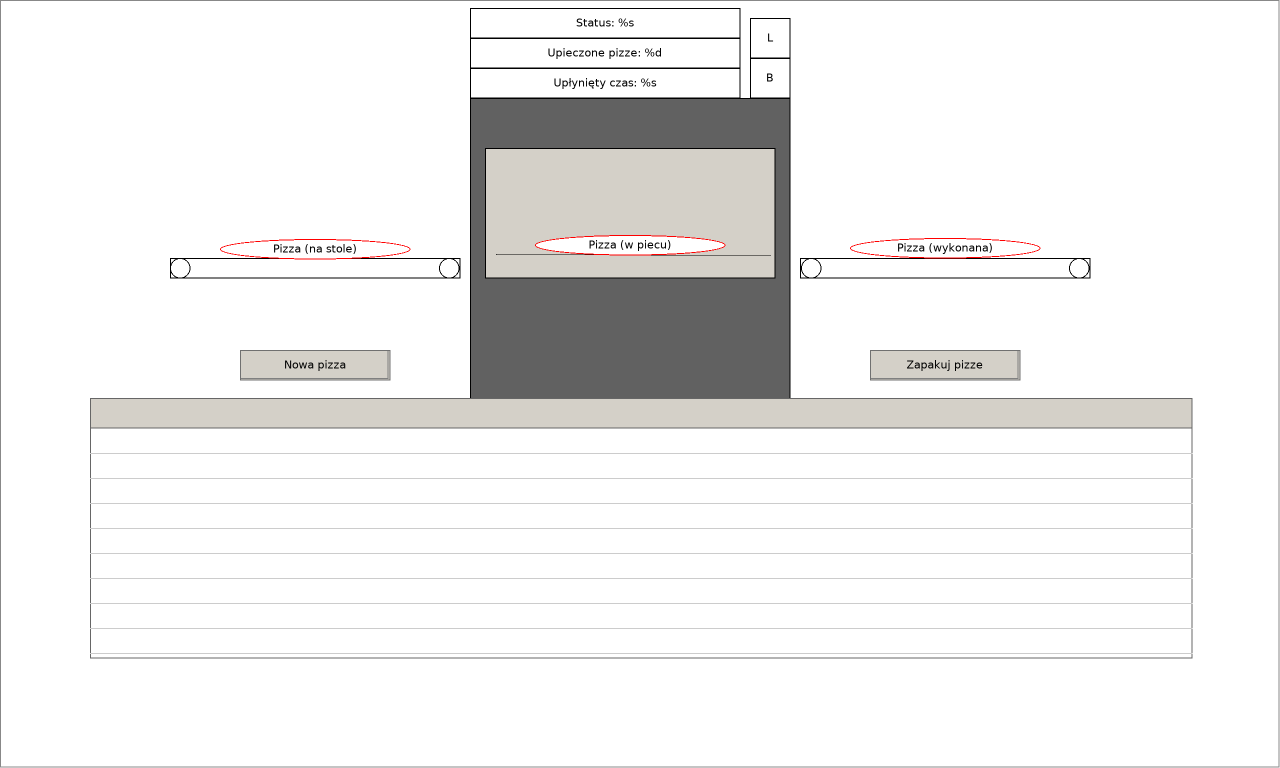
VISUALIZATION Visualization  // 1280x768
    Rectangle (470,98 320x480)
    Button (240,350 150x30), "Nowa pizza"
        tap MAIN.bLoadPizza
    Button (870,350 150x30), "Zapakuj pizze"
        tap MAIN.bRemovePizza
    Button (663,152 18x0)
    Rectangle (485,148 290x130)
    Rectangle (470,68 270x30), "Upłynięty czas: %s", text variable: MAIN.fbMyPizzaOven.fbMyTimer.ET
    RoundedRectangle (170,258 290x20)
    RoundedRectangle (800,258 290x20)
    Ellipse (850,238 190x20), "Pizza (wykonana)", invisible if: NOT MAIN.fbMyPizzaOven.stPizzaDone.bExist
    Ellipse (220,239 190x20), "Pizza (na stole)", invisible if: NOT MAIN.fbMyPizzaOven.stPizzaOnDeck.bExist
    Line (496,254) (770,255)
    Ellipse (535,235 190x20), "Pizza (w piecu)", invisible if: NOT MAIN.fbMyPizzaOven.stPizzaInOven.bExist
    RoundedRectangle (750,58 40x40), "B", colour toggle: MAIN.fbMyPizzaOven.bBuzzer
    RoundedRectangle (750,18 40x40), "L", colour toggle: MAIN.fbMyPizzaOven.bLight
    Rectangle (470,38 270x30), "Upieczone pizze: %d", text variable: MAIN.fbMyPizzaOven.iTotalPizzasCooked
    Ellipse (170,258 20x20)
    Ellipse (439,258 20x20)
    Rectangle (470,8 270x30), "Status: %s", text variable: MAIN.fbMyPizzaOven.sStateDesc
    Table (90,398 1102x260), data array: HMI_VARS.arrPizzaHistory
        p3854506369: HMI_VARS.arrPizzaHistory[INDEX].bExist
        p1892666644: HMI_VARS.arrPizzaHistory[INDEX].dtTimeEnteredOven
        p338671338: HMI_VARS.arrPizzaHistory[INDEX].dtTimeExitedOven
        p2170511999: HMI_VARS.arrPizzaHistory[INDEX].tTimeInOven
        p3723444502: HMI_VARS.arrPizzaHistory[INDEX].eType
        p2232123230: Czy pizza została wypieczona?
        p511219082: Data i godzina rozpoczęcia pieczenia pizzy
        p1755163831: Data i godzina zakończenia pieczenia pizzy
        p4092479075: Długość pieczenia pizzy
        p2237128397: Typ pizzy
    Ellipse (801,258 20x20)
    Ellipse (1069,258 20x20)
END_VISUALIZATION

(* stored: Version 1.1.0.1, ProductVersion 3.1.4024.11
   Visu Visualization: Id {67ce955f-c384-417c-86be-b3381fccb77a} *)
